TYPE Enviroment_Parameters :
STRUCT
END_STRUCT
END_TYPE

(* stored: Version 1.1.0.1, ProductVersion 3.1.4024.12
   DUT Enviroment_Parameters: Id {48760720-f476-4b9e-97b3-896a9e24eb50} *)
